VAR_GLOBAL
    gHostCmd  : ST_HostCmd;   // 上位机写入
    gPlcState : ST_PlcState;  // PLC 返回上位机
END_VAR

(* stored: Version 1.1.0.1, ProductVersion 3.1.4026.18
   GVL GVL_HMI: Id {12e7fd2d-dec6-4e6e-9cb0-a5b4830f8abe} *)
